// TIA Portal V16 export
// export: Created 2021-11-12T13:32:24.699909Z, ExportSetting WithDefaults, DisplayName Totally Integrated Automation Portal, DisplayVersion V16 Update 3, DisplayName TIA Portal Version Control Interface, DisplayVersion V16 Update 2, DisplayName TIA Portal Openness, DisplayVersion V16 Update 3, DisplayName SINAMICS Startdrive Advanced, DisplayVersion V16 Update 5, DisplayName SINAMICS Startdrive G130, G150, S120, S150, SINAMICS MV, S210, DisplayVersion V16 Update 5, DisplayName SINAMICS Startdrive G110M, G120, G120C, G120D, G120P, G115D, DisplayVersion V16 Update 5, DisplayName STEP 7 Professional, DisplayVersion V16 Update 3, DisplayName STEP 7 Safety, DisplayVersion V16, DisplayName WinCC UA Professional, DisplayVersion V16 Update 3
FUNCTION_BLOCK "StationKAS1"   // FB37, LAD
TITLE = Block for KASTO 1
{ S7_Optimized_Access := 'TRUE' }
VERSION : 0.1
// stored: AutoNumber true, IsIECCheckEnabled false, IsRetainMemResEnabled false, MemoryReserve 100, SetENOAutomatically false, UDAEnableTagReadback false
   VAR_INPUT
      IS_Inputs : "UDT_COMM_KAS1_CRS";   // Inputs from saws PLC
   END_VAR
   VAR_OUTPUT
      OS_Outputs : "UDT_COMM_CRS_KAS1";   // Outputs to saws PLC
   END_VAR
   VAR
      SF_Alarm1 : "STD_DI_Mon";
      SF_Alarm2 { S7_SetPoint := 'True'} : "STD_DI_Mon";
      SF_PartOk { S7_SetPoint := 'True'} : "STD_PartCounter";
      SF_PartNok { S7_SetPoint := 'True'} : "STD_PartCounter";
      SS_Edge : Array[0..15] of Bool;   // Edge evalution
   END_VAR
   VAR_TEMP   // added for the SCL form of the ladder/FBD networks
      _w1 : Bool;
      _w2 : Bool;
   END_VAR
BEGIN

REGION Network 1: ***************Alarms***************
END_REGION

REGION Network 2: Error in comunnication
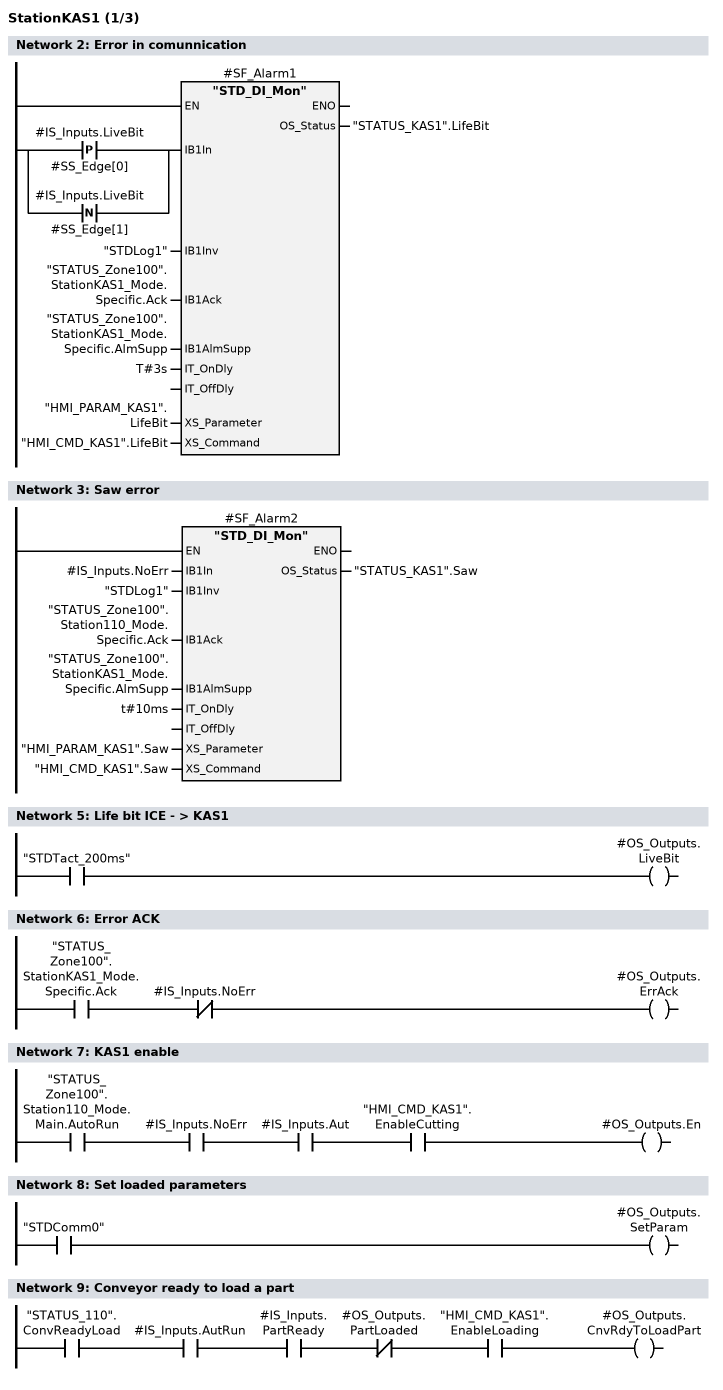
   RUNG wire#powerrail
      #SF_Alarm1(IB1In := wire#w1, IB1Inv := "STDLog1", IB1Ack := "STATUS_Zone100".StationKAS1_Mode.Specific.Ack, IB1AlmSupp := "STATUS_Zone100".StationKAS1_Mode.Specific.AlmSupp, IT_OnDly := T#3s, IT_OffDly :=, XS_Parameter := "HMI_PARAM_KAS1".LifeBit, XS_Command := "HMI_CMD_KAS1".LifeBit, OS_Status => "STATUS_KAS1".LifeBit)
   END_RUNG
   RUNG wire#powerrail
      P_Contact(operand := #IS_Inputs.LiveBit, bit := #SS_Edge[0])
   END_RUNG wire#w1
   RUNG wire#powerrail
      N_Contact(operand := #IS_Inputs.LiveBit, bit := #SS_Edge[1])
   END_RUNG wire#w1
   // the same network as SCL:
   #_w1 := #IS_Inputs.LiveBit AND NOT #SS_Edge[0];   // rising edge of #IS_Inputs.LiveBit
   #SS_Edge[0] := #IS_Inputs.LiveBit;
   #_w2 := NOT #IS_Inputs.LiveBit AND #SS_Edge[1];   // falling edge of #IS_Inputs.LiveBit
   #SS_Edge[1] := #IS_Inputs.LiveBit;
   #SF_Alarm1(IB1In := #_w1 OR #_w2,   // "STD_DI_Mon"
              IB1Inv := "STDLog1",
              IB1Ack := "STATUS_Zone100".StationKAS1_Mode.Specific.Ack,
              IB1AlmSupp := "STATUS_Zone100".StationKAS1_Mode.Specific.AlmSupp,
              IT_OnDly := T#3s,
              XS_Parameter := "HMI_PARAM_KAS1".LifeBit,
              XS_Command := "HMI_CMD_KAS1".LifeBit,
              OS_Status => "STATUS_KAS1".LifeBit);
END_REGION

REGION Network 3: Saw error
   RUNG wire#powerrail
      #SF_Alarm2(IB1In := #IS_Inputs.NoErr, IB1Inv := "STDLog1", IB1Ack := "STATUS_Zone100".Station110_Mode.Specific.Ack, IB1AlmSupp := "STATUS_Zone100".StationKAS1_Mode.Specific.AlmSupp, IT_OnDly := t#10ms, IT_OffDly :=, XS_Parameter := "HMI_PARAM_KAS1".Saw, XS_Command := "HMI_CMD_KAS1".Saw, OS_Status => "STATUS_KAS1".Saw)
   END_RUNG
   // the same network as SCL:
   #SF_Alarm2(IB1In := #IS_Inputs.NoErr,   // "STD_DI_Mon"
              IB1Inv := "STDLog1",
              IB1Ack := "STATUS_Zone100".Station110_Mode.Specific.Ack,
              IB1AlmSupp := "STATUS_Zone100".StationKAS1_Mode.Specific.AlmSupp,
              IT_OnDly := t#10ms,
              XS_Parameter := "HMI_PARAM_KAS1".Saw,
              XS_Command := "HMI_CMD_KAS1".Saw,
              OS_Status => "STATUS_KAS1".Saw);
END_REGION

REGION Network 4: ***************Remote***************
END_REGION

REGION Network 5: Life bit ICE - > KAS1
   RUNG wire#powerrail
      Contact( "STDTact_200ms" )
      Coil( #OS_Outputs.LiveBit )
   END_RUNG
   // the same network as SCL:
   #OS_Outputs.LiveBit := "STDTact_200ms";
END_REGION

REGION Network 6: Error ACK
   RUNG wire#powerrail
      Contact( "STATUS_Zone100".StationKAS1_Mode.Specific.Ack )
      I_Contact( #IS_Inputs.NoErr )
      Coil( #OS_Outputs.ErrAck )
   END_RUNG
   // the same network as SCL:
   #OS_Outputs.ErrAck := "STATUS_Zone100".StationKAS1_Mode.Specific.Ack AND NOT #IS_Inputs.NoErr;
END_REGION

REGION Network 7: KAS1 enable
   RUNG wire#powerrail
      Contact( "STATUS_Zone100".Station110_Mode.Main.AutoRun )
      Contact( #IS_Inputs.NoErr )
      Contact( #IS_Inputs.Aut )
      Contact( "HMI_CMD_KAS1".EnableCutting )
      Coil( #OS_Outputs.En )
   END_RUNG
   // the same network as SCL:
   #OS_Outputs.En := "STATUS_Zone100".Station110_Mode.Main.AutoRun AND #IS_Inputs.NoErr AND #IS_Inputs.Aut AND "HMI_CMD_KAS1".EnableCutting;
END_REGION

REGION Network 8: Set loaded parameters
   RUNG wire#powerrail
      Contact( "STDComm0" )
      Coil( #OS_Outputs.SetParam )
   END_RUNG
   // the same network as SCL:
   #OS_Outputs.SetParam := "STDComm0";
END_REGION

REGION Network 9: Conveyor ready to load a part
   RUNG wire#powerrail
      Contact( "STATUS_110".ConvReadyLoad )
      Contact( #IS_Inputs.AutRun )
      Contact( #IS_Inputs.PartReady )
      I_Contact( #OS_Outputs.PartLoaded )
      Contact( "HMI_CMD_KAS1".EnableLoading )
      Coil( #OS_Outputs.CnvRdyToLoadPart )
   END_RUNG
   // the same network as SCL:
   #OS_Outputs.CnvRdyToLoadPart := "STATUS_110".ConvReadyLoad AND #IS_Inputs.AutRun AND #IS_Inputs.PartReady AND NOT #OS_Outputs.PartLoaded AND "HMI_CMD_KAS1".EnableLoading;
END_REGION

REGION Network 10: Conveyor has loaded a part
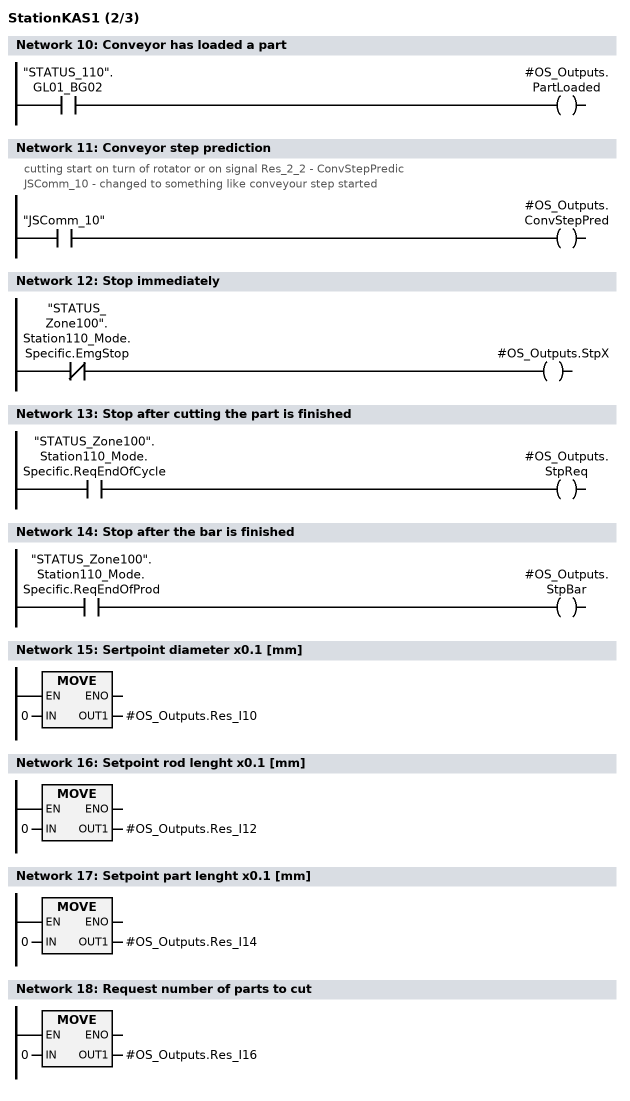
   RUNG wire#powerrail
      Contact( "STATUS_110".GL01_BG02 )
      Coil( #OS_Outputs.PartLoaded )
   END_RUNG
   // the same network as SCL:
   #OS_Outputs.PartLoaded := "STATUS_110".GL01_BG02;
END_REGION

REGION Network 11: Conveyor step prediction
   // cutting start on turn of rotator or on signal Res_2_2 - ConvStepPredic
   // JSComm_10 - changed to something like conveyour step started
   RUNG wire#powerrail
      Contact( "JSComm_10" )
      Coil( #OS_Outputs.ConvStepPred )
   END_RUNG
   // the same network as SCL:
   #OS_Outputs.ConvStepPred := "JSComm_10";
END_REGION

REGION Network 12: Stop immediately
   RUNG wire#powerrail
      I_Contact( "STATUS_Zone100".Station110_Mode.Specific.EmgStop )
      Coil( #OS_Outputs.StpX )
   END_RUNG
   // the same network as SCL:
   #OS_Outputs.StpX := NOT "STATUS_Zone100".Station110_Mode.Specific.EmgStop;
END_REGION

REGION Network 13: Stop after cutting the part is finished
   RUNG wire#powerrail
      Contact( "STATUS_Zone100".Station110_Mode.Specific.ReqEndOfCycle )
      Coil( #OS_Outputs.StpReq )
   END_RUNG
   // the same network as SCL:
   #OS_Outputs.StpReq := "STATUS_Zone100".Station110_Mode.Specific.ReqEndOfCycle;
END_REGION

REGION Network 14: Stop after the bar is finished
   RUNG wire#powerrail
      Contact( "STATUS_Zone100".Station110_Mode.Specific.ReqEndOfProd )
      Coil( #OS_Outputs.StpBar )
   END_RUNG
   // the same network as SCL:
   #OS_Outputs.StpBar := "STATUS_Zone100".Station110_Mode.Specific.ReqEndOfProd;
END_REGION

REGION Network 15: Sertpoint diameter x0.1 [mm]
   RUNG wire#powerrail
      Move(in := 0, out1 => #OS_Outputs.Res_I10)
   END_RUNG
   // the same network as SCL:
   #OS_Outputs.Res_I10 := 0;
END_REGION

REGION Network 16: Setpoint rod lenght x0.1 [mm]
   RUNG wire#powerrail
      Move(in := 0, out1 => #OS_Outputs.Res_I12)
   END_RUNG
   // the same network as SCL:
   #OS_Outputs.Res_I12 := 0;
END_REGION

REGION Network 17: Setpoint part lenght x0.1 [mm]
   RUNG wire#powerrail
      Move(in := 0, out1 => #OS_Outputs.Res_I14)
   END_RUNG
   // the same network as SCL:
   #OS_Outputs.Res_I14 := 0;
END_REGION

REGION Network 18: Request number of parts to cut
   RUNG wire#powerrail
      Move(in := 0, out1 => #OS_Outputs.Res_I16)
   END_RUNG
   // the same network as SCL:
   #OS_Outputs.Res_I16 := 0;
END_REGION

REGION Network 19: *************** Status ***************
END_REGION

REGION Network 20: Number of parts which length is correct
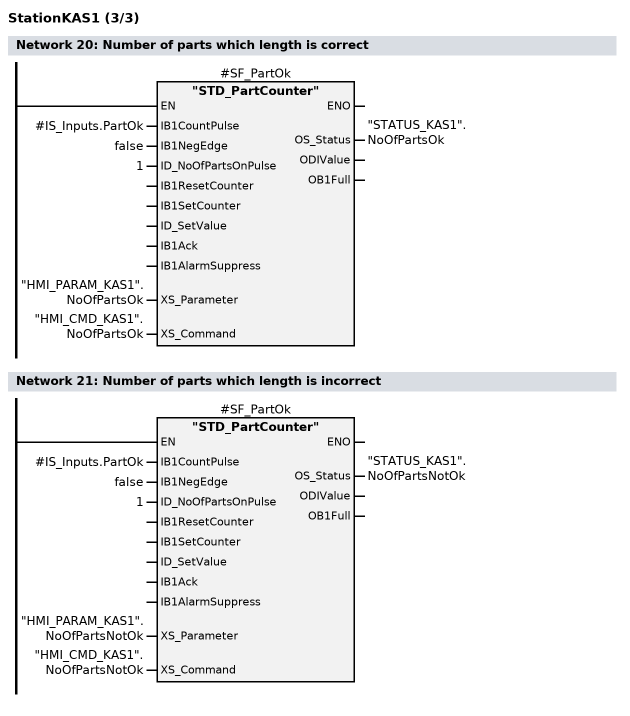
   RUNG wire#powerrail
      #SF_PartOk(IB1CountPulse := #IS_Inputs.PartOk, IB1NegEdge := false, ID_NoOfPartsOnPulse := 1, IB1ResetCounter :=, IB1SetCounter :=, ID_SetValue :=, IB1Ack :=, IB1AlarmSuppress :=, XS_Parameter := "HMI_PARAM_KAS1".NoOfPartsOk, XS_Command := "HMI_CMD_KAS1".NoOfPartsOk, OS_Status => "STATUS_KAS1".NoOfPartsOk, ODIValue =>, OB1Full =>)
   END_RUNG
   // the same network as SCL:
   #SF_PartOk(IB1CountPulse := #IS_Inputs.PartOk,   // "STD_PartCounter"
              IB1NegEdge := false,
              ID_NoOfPartsOnPulse := 1,
              XS_Parameter := "HMI_PARAM_KAS1".NoOfPartsOk,
              XS_Command := "HMI_CMD_KAS1".NoOfPartsOk,
              OS_Status => "STATUS_KAS1".NoOfPartsOk);
END_REGION

REGION Network 21: Number of parts which length is incorrect
   RUNG wire#powerrail
      #SF_PartOk(IB1CountPulse := #IS_Inputs.PartOk, IB1NegEdge := false, ID_NoOfPartsOnPulse := 1, IB1ResetCounter :=, IB1SetCounter :=, ID_SetValue :=, IB1Ack :=, IB1AlarmSuppress :=, XS_Parameter := "HMI_PARAM_KAS1".NoOfPartsNotOk, XS_Command := "HMI_CMD_KAS1".NoOfPartsNotOk, OS_Status => "STATUS_KAS1".NoOfPartsNotOk, ODIValue =>, OB1Full =>)
   END_RUNG
   // the same network as SCL:
   #SF_PartOk(IB1CountPulse := #IS_Inputs.PartOk,   // "STD_PartCounter"
              IB1NegEdge := false,
              ID_NoOfPartsOnPulse := 1,
              XS_Parameter := "HMI_PARAM_KAS1".NoOfPartsNotOk,
              XS_Command := "HMI_CMD_KAS1".NoOfPartsNotOk,
              OS_Status => "STATUS_KAS1".NoOfPartsNotOk);
END_REGION
END_FUNCTION_BLOCK
